{attribute 'qualified_only'}
VAR_GLOBAL CONSTANT
	
END_VAR

(* stored: Version 1.1.0.1, ProductVersion 3.1.4024.14
   GVL GVL_CONSTANT: Id {a2c7890f-3858-4b75-847c-a1850ca751f3} *)
